// SIMATIC S7-200 project (STEP 7-Micro/WIN), CPU 226 REL 02.01

SYMBOL_TABLE USER1
Start            I0.0
AStop            I0.1
Motor1           Q0.0
Motor2           Q0.1
Motor3           Q0.2
END_SYMBOL_TABLE

ORGANIZATION_BLOCK MAIN:OB1
TITLE=PROGRAM COMMENTS
BEGIN
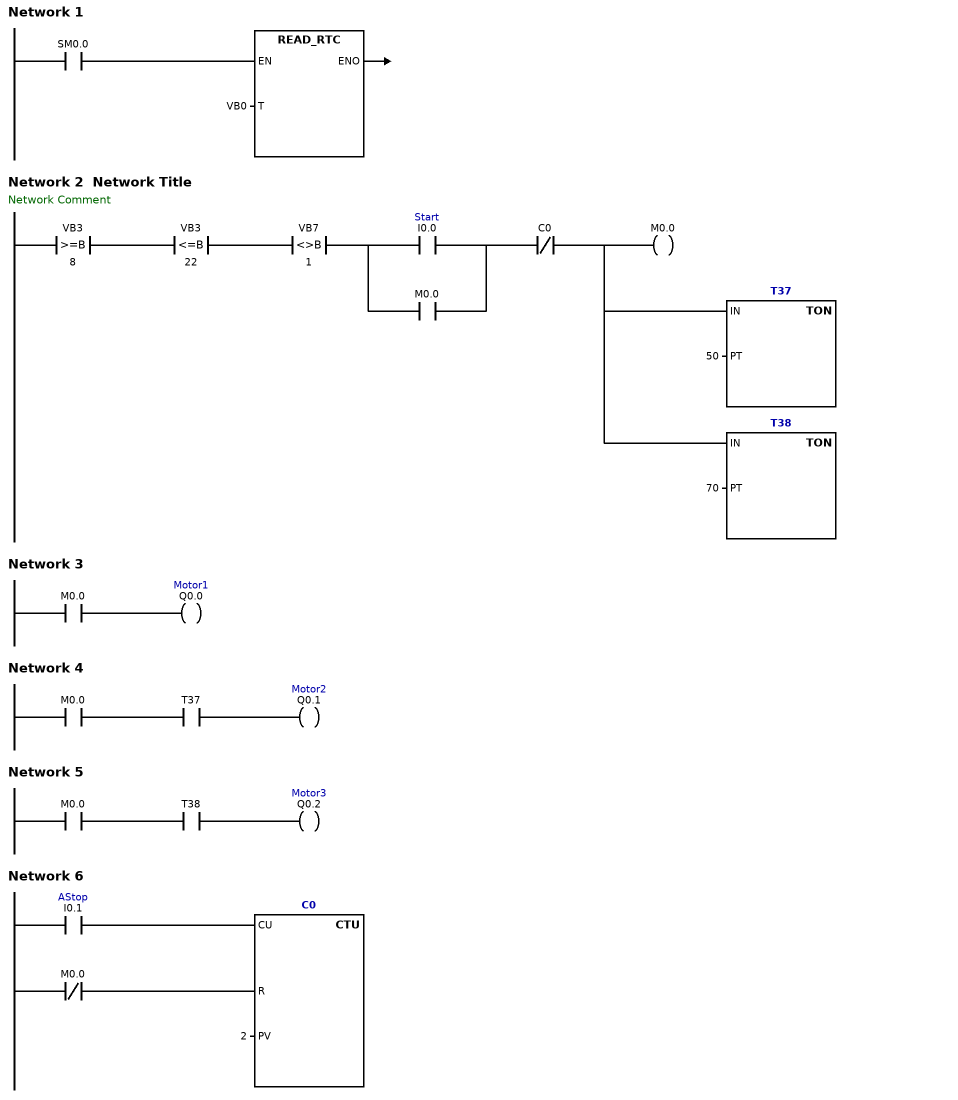
Network 1
LD     SM0.0
TODR   VB0
Network 2 // Network Title
// Network Comment
LDB>=  VB3, 8
AB<=   VB3, 22
AB<>   VB7, 1
LD     Start:I0.0
O      M0.0
ALD
AN     C0
=      M0.0
TON    T37, 50
TON    T38, 70
Network 3
LD     M0.0
=      Motor1:Q0.0
Network 4
LD     M0.0
A      T37
=      Motor2:Q0.1
Network 5
LD     M0.0
A      T38
=      Motor3:Q0.2
Network 6
LD     AStop:I0.1
LDN    M0.0
CTU    C0, 2
END_ORGANIZATION_BLOCK
